// TIA Portal V17 export
// export: Created 2023-09-10T16:27:52.8768317Z, ExportSetting WithDefaults, DisplayName Totally Integrated Automation Portal, DisplayVersion V17, DisplayName TIA Portal Openness, DisplayVersion V17, DisplayName TIA Portal Version Control Interface, DisplayVersion V17, DisplayName STEP 7 Professional, DisplayVersion V17, DisplayName STEP 7 Safety, DisplayVersion V17, DisplayName WinCC Advanced, DisplayVersion V17
DATA_BLOCK "machineData"   // DB1
{ S7_Optimized_Access := 'TRUE' }
VERSION : 0.1
// stored: AutoNumber true, DBAccessibleFromOPCUA true, IsOnlyStoredInLoadMemory false, IsRetainMemResEnabled false, IsWriteProtectedInAS false, MemoryReserve 100
   VAR
      encoderTurn : DInt;
      reqVelocity : Real;
      encoderValue : Int;
   END_VAR
   VAR RETAIN
      machinePosition : DInt;
   END_VAR
   VAR
      direction : Bool;
   END_VAR
   VAR RETAIN
      lastEncoderValue : DInt;
      lastMachinePosition : DInt;
   END_VAR
BEGIN
END_DATA_BLOCK
